// TIA Portal V17 export
// export: Created 2025-08-28T07:22:31.6285826Z, ExportSetting WithDefaults, DisplayName Totally Integrated Automation Portal, DisplayVersion V17, DisplayName TIA Portal Openness, DisplayVersion V17, DisplayName TIA Portal Version Control Interface, DisplayVersion V17, DisplayName STEP 7 Professional, DisplayVersion V17, DisplayName STEP 7 Safety, DisplayVersion V17, DisplayName WinCC Advanced, DisplayVersion V17
VAR_GLOBAL   // PLC tag table "默认变量表"
   "1号计量泵运行" AT %I0.0 : Bool;
   "2号计量泵运行" AT %I0.2 : Bool;
   "3号计量泵运行" AT %I0.4 : Bool;
   "1号计量泵故障" AT %I0.1 : Bool;
   "2号计量泵故障" AT %I0.3 : Bool;
   "3号计量泵故障" AT %I0.5 : Bool;
   "1号药池电动阀开到位" AT %I0.6 : Bool;
   "2号药池电动阀开到位" AT %I1.0 : Bool;
   "1号药池电动阀关到位" AT %I0.7 : Bool;
   "2号药池电动阀关到位" AT %I1.1 : Bool;
   新旧电柜控制切换 AT %I1.2 : Bool;
   本电柜和中控控制切换 AT %I1.3 : Bool;
   "1号泵流量反馈" AT %IW96 : Int;
   "2号泵流量反馈" AT %IW98 : Int;
   "3号泵流量反馈" AT %IW100 : Int;
   "1号罐液位" AT %IW104 : Int;
   "2号罐液位" AT %IW106 : Int;
   紧急停机 AT %I1.4 : Bool;
   "1号计量泵启停" AT %Q0.0 : Bool;
   "2号计量泵启停" AT %Q0.1 : Bool;
   "3号计量泵启停" AT %Q0.2 : Bool;
   "1号药池电动阀打开关闭" AT %Q0.3 : Bool;
   "2号药池电动阀打开关闭" AT %Q0.4 : Bool;
   "1号泵流量控制" AT %QW112 : Int;
   "2号泵流量控制" AT %QW114 : Int;
   "3号泵流量控制" AT %QW116 : Int;
   ET AT %MD0 : Time;
END_VAR
